PROGRAM MAIN
VAR
	fbLiquidTank : FB_Tank; 	

	bFillButton : BOOL;
	bDrainButton : BOOL;
END_VAR

fbLiquidTank(bIsFillButtonPressed := bFillButton, bIsDrainButtonPressed := bDrainButton);

END_PROGRAM

(* stored: Version 1.1.0.1, ProductVersion 3.1.4024.12
   POU MAIN: Id {cd576b26-1fdb-4b4f-8944-02a8451659e2}, SpecialFunc None *)
